IsRegValid:=FALSE;

// Температуры
// Проверка температур
FOR I:=0 TO NUM_TEMPS-1 DO
	IF (pr^.TEMPS[I] < 0) OR (pr^.TEMPS[I] > T_CRITICALS[I]) THEN
		RETURN;
	END_IF
END_FOR

// Температура чиллера
IF (pr^.T_CHIL < 0) OR (pr^.T_CHIL > T_CHIL_CRITICAL) THEN
	RETURN;
END_IF

// Смещение 1-го полупериода
IF pr^.Period.Offsets[0] = pr^.Period.Offsets[1] THEN
	RETURN;
END_IF

// Смещение 2-го полупериода
IF ABS (pr^.Period.Offsets[0] - pr^.Period.Offsets[1]) > WORK_SIZE THEN
	RETURN;
END_IF

// Проценты полупериодов
IF pr^.Period.Per_FirstHP < ASDA_HP_MIN OR pr^.Period.Per_FirstHP > ASDA_HP_MAX THEN
	RETURN;
END_IF

// Проценты импульсов
IF pr^.Period.Per_Pulses[0] < ASDA_PULSE_MIN OR pr^.Period.Per_Pulses[0] > ASDA_PULSE_MAX THEN
	RETURN;
END_IF

IF pr^.Period.Per_Pulses[1] < ASDA_PULSE_MIN OR pr^.Period.Per_Pulses[1] > ASDA_PULSE_MAX THEN
	RETURN;
END_IF

// Проценты уровня
IF pr^.Period.Per_Levels[0] < ASDA_LEVEL_MIN OR pr^.Period.Per_Levels[0] > ASDA_LEVEL_MAX THEN
	RETURN;
END_IF

IF pr^.Period.Per_Levels[1] < ASDA_LEVEL_MIN OR pr^.Period.Per_Levels[1] > ASDA_LEVEL_MAX THEN
	RETURN;
END_IF

// Скорость заготовки
IF pr^.Speed < SPEED_MIN OR pr^.Speed >= SPEED_MAX THEN
	RETURN;
END_IF

// Длина заготовки
IF pr^.Length < LEN_MIN OR pr^.Length > LEN_MAX THEN
	RETURN;
END_IF

// Производительность
IF pr^.Qm < QM_MIN OR pr^.Qm > QM_MAX THEN
	RETURN;
END_IF

IsRegValid:=TRUE;

END_FUNCTION

// Device/Application/SRC/AsdaSetPeriod
PROGRAM AsdaSetPeriod
VAR
	dRep		: DINT;
	wSpeeds		: ARRAY [0..1] OF WORD;			// обороты в мин
	wAccs		: ARRAY [0..3] OF WORD;			// обороты в мин
	wDels		: ARRAY [0..1] OF WORD;			// милисекунды
	dOffsets	: ARRAY [0..1] OF DINT;
	dist		: REAL;
	tPeriod		: REAL;			
	tHalfs		: ARRAY [0..1] OF REAL;
	tPulses		: ARRAY [0..1] OF REAL;
	tLevels		: ARRAY [0..1] OF REAL;
	tAccs		: ARRAY [0..1] OF REAL;
	midSpeeds	: ARRAY [0..1] OF REAL;
	vSpeeds		: ARRAY [0..1] OF REAL;
END_VAR


CASE Asda.SelButton OF

sbPeriod:	// УСТАНОВКА ПАРАМЕТРОВ ПЕРИОДА

	// 1. Сначала записать положение реперной точки P6-01, адрес 16х0602
	dRep:=REAL_TO_DINT (REP_MM * PUU_PER_MM);
	QueuePushReg (ADR (COM1_PRG.WR_REGS), ADR_ASDA, 16#0602, ADR (dRep), 2);			// Р6-01 Положение реперной точки

	// 2. Запись перемещения 1-го полупериода, т.к. оно используется при вычислении следующих параметров
	dOffsets[0]:=REAL_TO_DINT (REG_W.Period.Offsets[0] * PUU_PER_MM);
	QueuePushReg (ADR (COM1_PRG.WR_REGS), ADR_ASDA, 16#062A, ADR (dOffsets[0]), 2);	// Р6-21 Смещение 1-го полупериода рабочее
	QueuePushReg (ADR (COM1_PRG.WR_REGS), ADR_ASDA, 16#063A, ADR (dOffsets[0]), 2);	// Р6-29 Смещение 1-го полупериода для ШАГА позиционирования 14 (ручное перемещение)

	// Запись перемещения 2-го полупериода, т.к. оно используется при вычислении следующих параметров
	dOffsets[1]:=REAL_TO_DINT (REG_W.Period.Offsets[1] * PUU_PER_MM);
	QueuePushReg (ADR (COM1_PRG.WR_REGS), ADR_ASDA, 16#062E, ADR (dOffsets[1]), 2);	// Р6-23 Смещение 2-го полупериода
	QueuePushReg (ADR (COM1_PRG.WR_REGS), ADR_ASDA, 16#063E, ADR (dOffsets[1]), 2);	// Р6-31 Смещение 2-го полупериода для шага позиционирования 15 (ручное перемещение)

	// Время периода в секундах
	tPeriod:= 1 / REG_W.Period.Freq;
	
	// Времена полупериодов в секундах
	tHalfs[0]:=tPeriod * REG_W.Period.Per_FirstHP / 100;
	tHalfs[1]:=tPeriod - tHalfs[0];
	
	// Времена импульсов в секундах
	tPulses[0]:=tHalfs[0] * REG_W.Period.Per_Pulses[0] / 100;
	tPulses[1]:=tHalfs[1] * REG_W.Period.Per_Pulses[1] / 100;
	
	// Фронты полупериодов (импульсов) в секундах - Длина импульса минус длина уровня, делённая на 2
	tAccs[0]:=tPulses[0] * (100 - REG_W.Period.Per_Levels[0]) / 200;
	tAccs[1]:=tPulses[1] * (100 - REG_W.Period.Per_Levels[1]) / 200;
	
	// Уровни полупериодов
	tLevels[0]:=tPulses[0] * REG_W.Period.Per_Levels[0] / 100;
	tLevels[1]:=tPulses[1] * REG_W.Period.Per_Levels[1] / 100;
	
	// Пройденный путь в мм
	dist:=ABS (REG_W.Period.Offsets[0] - REG_W.Period.Offsets[1]);
	
	// Средние скорости в мм/сек
	midSpeeds[0]:=dist / tPulses[0];
	midSpeeds[1]:=dist / tPulses[1];
	
	// Расчётные скорости в мм/сек
	vSpeeds[0]:=midSpeeds[0] * (2 * tAccs[0] + tLevels[0]) / (tAccs[0] + tLevels[0]);
	vSpeeds[1]:=midSpeeds[1] * (2 * tAccs[1] + tLevels[1]) / (tAccs[1] + tLevels[1]);
		
	// Пересчёт скорости, данные - l оборот => 5 мм перемещения
	// 5 мм/сек = 1 об/сек =>
	wSpeeds[0]:=REAL_TO_WORD (vSpeeds[0] * 60 * 10 / 5);	// Получили в об/мин (Нужно умножить на 10, т.к. в сервоприводе единица измерения скорости 0.1 об/мин)
	wSpeeds[1]:=REAL_TO_WORD (vSpeeds[1] * 60 * 10 / 5);	// Получили в об/мин

	// Пересчёт фронт и спада относительно скорости wSpeeds[0]
	wAccs[0]:=REAL_TO_WORD (tAccs[0] * 3000 * 1000 / wSpeeds[0]);	
	wAccs[1]:=REAL_TO_WORD (tAccs[0] * 3000 * 1000 / wSpeeds[0]);
	wAccs[2]:=REAL_TO_WORD (tAccs[1] * 3000 * 1000 / wSpeeds[1]);
	wAccs[3]:=REAL_TO_WORD (tAccs[1] * 3000 * 1000 / wSpeeds[1]);
	
	// Задержки в миллисекундах
	wDels[0]:=REAL_TO_WORD ((tHalfs[0] - tPulses[0]) * 1000.0);
	wDels[1]:=REAL_TO_WORD ((tHalfs[1] - tPulses[1]) * 1000.0);

	// Запись	
	QueuePushReg (ADR (COM1_PRG.WR_REGS), ADR_ASDA, 16#0528, ADR (wAccs[0]), 1);		// Р5-20 Фронт 1-го полупериода
	QueuePushReg (ADR (COM1_PRG.WR_REGS), ADR_ASDA, 16#052A, ADR (wAccs[1]), 1);		// Р5-21 Спад 1-го полупериода 
	QueuePushReg (ADR (COM1_PRG.WR_REGS), ADR_ASDA, 16#052C, ADR (wAccs[2]), 1);		// Р5-22 Фронт 2-го полупериода
	QueuePushReg (ADR (COM1_PRG.WR_REGS), ADR_ASDA, 16#052E, ADR (wAccs[3]), 1);		// Р5-23 Спад 2-го полупериода 

	QueuePushReg (ADR (COM1_PRG.WR_REGS), ADR_ASDA, 16#0578, ADR (wSpeeds[0]), 1);		// Р5-60 Скорость 1-го полупериода
	QueuePushReg (ADR (COM1_PRG.WR_REGS), ADR_ASDA, 16#057A, ADR (wSpeeds[1]), 1);		// Р5-61 Скорость 2-го полупериода 

	QueuePushReg (ADR (COM1_PRG.WR_REGS), ADR_ASDA, 16#0550, ADR (wDels[0]), 1);		// Р5-40 Задержка 1-го полупериода
	QueuePushReg (ADR (COM1_PRG.WR_REGS), ADR_ASDA, 16#0552, ADR (wDels[1]), 1);		// Р5-41 Задержка 2-го полупериода

// Команда Homing
sbHoming: AddWriteCmd (wCmd:=wcAsda_Homing);
	
// Движение вперёд
sbForward: AddWriteCmd (wCmd:=wcAsda_Forward);

// Движение назад
sbBackward: AddWriteCmd (wCmd:=wcAsda_Backward);

// Парковка
sbParking: AddWriteCmd (wCmd:=wcAsda_Parking);

// Работа (пульсирование)
sbWorking: AddWriteCmd (wCmd:=wcAsda_Working);
	
END_CASE

Asda.SelButton:=sbNo;
Asda.bCmd:=FALSE;

END_PROGRAM

// Device/Application/SRC_AUX/SWAP_BYTES
FUNCTION SWAP_BYTES : WORD
VAR_INPUT
	wValue : WORD;
END_VAR
VAR
END_VAR


SWAP_BYTES := SHL (wValue, 8) OR SHR (wValue, 8);

END_FUNCTION

// Device/Application/SRC/SET_FRAME_INDEX_EX
FUNCTION SET_FRAME_INDEX_EX : BYTE
VAR_INPUT
	Index : BYTE;
END_VAR
VAR
END_VAR
VAR // added by the converter: edge detectors and wires of the graphical bodies
    _w1 : ANY;
END_VAR

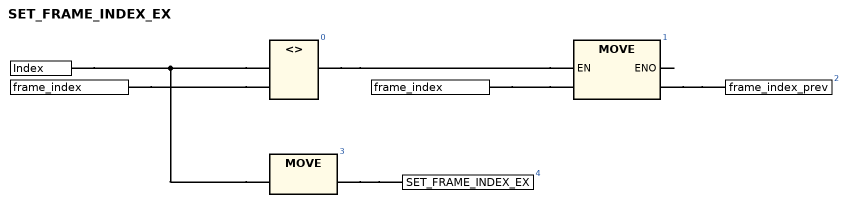
IF Index <> frame_index THEN _w1 := frame_index; END_IF
frame_index_prev := _w1;
SET_FRAME_INDEX_EX := Index;

END_FUNCTION

// Device/Application/SRC_AUX/BYTES_FROM_DINT
FUNCTION BYTES_FROM_DINT : BOOL
VAR_INPUT
	pBytes	: POINTER TO BYTE;
	iDint	: DINT;
END_VAR
VAR
	pB		: POINTER TO BYTE;
END_VAR

BYTES_FROM_DINT:=TRUE;

pB:=ADR(iDint);

pBytes[0]:=pB[1];
pBytes[1]:=pB[0];
pBytes[2]:=pB[3];
pBytes[3]:=pB[2];

END_FUNCTION

// Device/Application/SRC/MERGE_RGB
FUNCTION MERGE_RGB : DWORD
VAR_INPUT
	clR	: BYTE;
	clG	: BYTE;
	clB	: BYTE;
END_VAR
VAR
END_VAR

MERGE_RGB:=BYTE_TO_DWORD(255);
MERGE_RGB:=SHL(MERGE_RGB,8);
MERGE_RGB:=MERGE_RGB OR BYTE_TO_DWORD(clR);
MERGE_RGB:=SHL(MERGE_RGB,8);
MERGE_RGB:=MERGE_RGB OR BYTE_TO_DWORD(clG);
MERGE_RGB:=SHL(MERGE_RGB,8);
MERGE_RGB:=MERGE_RGB OR BYTE_TO_DWORD(clB);

END_FUNCTION

// Device/Application/SRC_FILE/WRITE_OPTIONS
FUNCTION WRITE_OPTIONS : BOOL
VAR_INPUT
	Show	: BOOL;
END_VAR
VAR
	hFile	: SysFile.RTS_IEC_HANDLE;	
	Result	: SysFile.RTS_IEC_RESULT;
	rSize	: __XWORD;
	wrBytes	: __XWORD;
	
END_VAR

WRITE_OPTIONS:=FALSE;
// Создаём новый файл
hFile:=SysFileOpen (OPTIONSFILE,SysFile.AM_WRITE, ADR (Result));
IF Result <> 0 THEN
	RETURN;
END_IF

rSize:=SIZEOF (TSetts);

wrBytes:=SysFileWrite(hFile, ADR (Setts), rSize, ADR (Result));
IF (Result=0) AND (wrBytes=rSize) THEN
	WRITE_OPTIONS:=TRUE;
END_IF

SysFileClose (hFile);

END_FUNCTION

// Device/Application/SRC_AUX/HiWord
FUNCTION HiWord : WORD
VAR_INPUT
	dValue	: DINT;
END_VAR	
VAR
	pW		: POINTER TO WORD;
END_VAR

pW:= ADR (dValue);
HiWord:=pW[1];

END_FUNCTION

// Device/Application/SRC_FILE/READ_OPTIONS
FUNCTION READ_OPTIONS : BOOL
VAR
	hFile	: SysFile.RTS_IEC_HANDLE;	
	Result	: SysFile.RTS_IEC_RESULT;
	fSize	: __XWORD;
	rSize	: __XWORD;
	rdBytes	: __XWORD;
	rdSetts	: TSetts;
	
END_VAR

READ_OPTIONS:=FALSE;

rSize:=SIZEOF(TSetts);

hFile:=SysFileOpen (OPTIONSFILE, SysFile.AM_READ, ADR (Result));
IF Result <> 0 THEN
	RETURN;
END_IF

//  Файл существует, проверяем размер файла
fSize:=SysFileGetSizeByHandle (hFile, ADR (Result));
IF Result <> 0 OR fSize <> rSize THEN
	SysFileClose(hFile);
	RETURN;	
END_IF

rdBytes:=SysFileRead(hFile, ADR (rdSetts), rSize, ADR (Result));	
IF Result = 0 AND rdBytes = rSize THEN
	Setts:=rdSetts;
	READ_OPTIONS:=TRUE;
END_IF

SysFileClose(hFile);

END_FUNCTION

// Device/Application/SRC_AUX/LoWord
FUNCTION LoWord : WORD
VAR_INPUT
	dValue	: DINT;
END_VAR
VAR
	pW		: POINTER TO WORD;
END_VAR

pW:= ADR (dValue);
LoWord:=pW[0];

END_FUNCTION

// Device/Application/SRC_AUX/LoByte
FUNCTION LoByte : BYTE
VAR_INPUT
	W	: WORD;
END_VAR
VAR
END_VAR

LoByte:=WORD_TO_BYTE (W AND 16#FF);

END_FUNCTION

// Device/Application/SRC_AUX/HiByte
FUNCTION HiByte : BYTE
VAR_INPUT
	W : WORD;
END_VAR
VAR
END_VAR

HiByte:= WORD_TO_BYTE (SHR (W, 8) AND 16#FF);

END_FUNCTION

// Device/Application/SRC_AUX/IsRegTempersValid
FUNCTION IsRegTempersValid : BOOL
VAR_INPUT
	pr : POINTER TO TReg;
	
END_VAR
VAR
	I: INT;
END_VAR

IsRegTempersValid:=FALSE;

// Температуры
// Проверка температур уставок (без TEMPS[7])	
FOR I:=0 TO NUM_TEMPS-2 DO
	
	// Если задана температура ниже температуры запуска приводов или выше критической 
	IF (pr^.TEMPS[I] < Setts.T_ZAP[I]) OR (pr^.TEMPS[I] > T_CRITICALS[I]) THEN
		RETURN;
	END_IF
	
END_FOR

IsRegTempersValid:=TRUE;

END_FUNCTION

// Device/Application/SRC_AUX/BYTES_FROM_INT
FUNCTION BYTES_FROM_INT : BOOL
VAR_INPUT
	pBytes	: POINTER TO BYTE;
	vInt	: INT;
END_VAR
VAR
	pB		: POINTER TO BYTE;
END_VAR

BYTES_FROM_INT:=TRUE;

pB:=ADR(vInt);
pBytes[0]:=pB[1];
pBytes[1]:=pB[0];

END_FUNCTION

// Device/Application/Visu/VIS_AUX
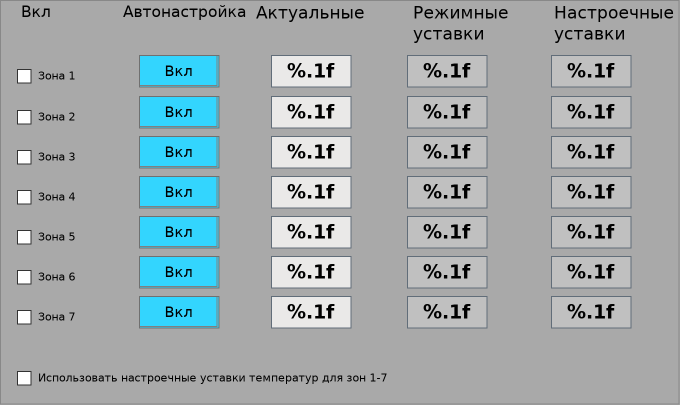
VISUALIZATION VIS_AUX  // 680x405
    Checkbox (15,55 120x42), "Зона 1", variable: Dvp.T_Enables.0
    Checkbox (15,96 120x42), "Зона 2", variable: Dvp.T_Enables.1
    Checkbox (15,136 120x42), "Зона 3", variable: Dvp.T_Enables.2
    Checkbox (15,176 120x42), "Зона 4", variable: Dvp.T_Enables.3
    Checkbox (15,216 120x42), "Зона 5", variable: Dvp.T_Enables.4
    Checkbox (15,256 120x42), "Зона 6", variable: Dvp.T_Enables.5
    Checkbox (15,296 120x42), "Зона 7", variable: Dvp.T_Enables.6
    Label (18,1 63x24), "Вкл"
    Label (120,1 129x28), "Автонастройка"
    Button (139,55 80x32), "Вкл", colour toggle: Dvp.Auto_IN.0
        OnMouseClick: execute { Dvp.Auto_OUT.0:=TRUE; }
    Button (139,96 80x32), "Вкл", colour toggle: Dvp.Auto_IN.1
        OnMouseClick: execute { Dvp.Auto_OUT.1:=TRUE; }
    Button (139,136 80x32), "Вкл", colour toggle: Dvp.Auto_IN.2
        OnMouseClick: execute { Dvp.Auto_OUT.2:=TRUE; }
    Button (139,176 80x32), "Вкл", colour toggle: Dvp.Auto_IN.3
        OnMouseClick: execute { Dvp.Auto_OUT.3:=TRUE; }
    Button (139,216 80x32), "Вкл", colour toggle: Dvp.Auto_IN.4
        OnMouseClick: execute { Dvp.Auto_OUT.4:=TRUE; }
    Button (139,256 80x32), "Вкл", colour toggle: Dvp.Auto_IN.5
        OnMouseClick: execute { Dvp.Auto_OUT.5:=TRUE; }
    Button (139,296 80x32), "Вкл", colour toggle: Dvp.Auto_IN.6
        OnMouseClick: execute { Dvp.Auto_OUT.6:=TRUE; }
    Checkbox (15,357 589x42), "Использовать настроечные уставки температур для зон 1-7", variable: zd_selector
    RoundedRectangle (407,55 80x32), "%.1f", text variable: REG_W.TEMPS[0], colour toggle: NOT zd_selector
    RoundedRectangle (407,96 80x32), "%.1f", text variable: REG_W.TEMPS[1], colour toggle: NOT zd_selector
    RoundedRectangle (407,136 80x32), "%.1f", text variable: REG_W.TEMPS[2], colour toggle: NOT zd_selector
    RoundedRectangle (407,176 80x32), "%.1f", text variable: REG_W.TEMPS[3], colour toggle: NOT zd_selector
    RoundedRectangle (407,216 80x32), "%.1f", text variable: REG_W.TEMPS[4], colour toggle: NOT zd_selector
    RoundedRectangle (407,256 80x32), "%.1f", text variable: REG_W.TEMPS[5], colour toggle: NOT zd_selector
    RoundedRectangle (407,296 80x32), "%.1f", text variable: REG_W.TEMPS[6], colour toggle: NOT zd_selector
    Label (410,1 107x49), "Режимные уставки"
    RoundedRectangle (551,55 80x32), "%.1f", text variable: zd_temps[0], colour toggle: zd_selector
        OnMouseClick: write the text variable via VisuDialogs.Numpad, min T_MINS_ZAD[6], max T_MAXS_ZAD[6], title "ТЕМПЕРАТУРА 7 ЗОНЫ"
    RoundedRectangle (551,96 80x32), "%.1f", text variable: zd_temps[1], colour toggle: zd_selector
        OnMouseClick: write the text variable via VisuDialogs.Numpad, min T_MINS_ZAD[0], max T_MAXS_ZAD[0]
    RoundedRectangle (551,136 80x32), "%.1f", text variable: zd_temps[2], colour toggle: zd_selector
        OnMouseClick: write the text variable via VisuDialogs.Numpad, min T_MINS_ZAD[0], max T_MAXS_ZAD[0]
    RoundedRectangle (551,176 80x32), "%.1f", text variable: zd_temps[3], colour toggle: zd_selector
        OnMouseClick: write the text variable via VisuDialogs.Numpad, min T_MINS_ZAD[0], max T_MAXS_ZAD[0]
    RoundedRectangle (551,216 80x32), "%.1f", text variable: zd_temps[4], colour toggle: zd_selector
        OnMouseClick: write the text variable via VisuDialogs.Numpad, min T_MINS_ZAD[0], max T_MAXS_ZAD[0]
    RoundedRectangle (551,256 80x32), "%.1f", text variable: zd_temps[5], colour toggle: zd_selector
        OnMouseClick: write the text variable via VisuDialogs.Numpad, min T_MINS_ZAD[0], max T_MAXS_ZAD[0]
    RoundedRectangle (551,296 80x32), "%.1f", text variable: zd_temps[6], colour toggle: zd_selector
        OnMouseClick: write the text variable via VisuDialogs.Numpad, min T_MINS_ZAD[0], max T_MAXS_ZAD[0]
    Label (551,1 127x47), "Настроечные уставки"
    RoundedRectangle (271,55 80x32), "%.1f", text variable: Dvp.T_Actuals[0], colour variable: Dvp.FillColors[0]
        p3450524324: Dvp.FrameColors[0]
    RoundedRectangle (271,96 80x32), "%.1f", text variable: Dvp.T_Actuals[1], colour variable: Dvp.FillColors[1]
        p3450524324: Dvp.FrameColors[1]
    RoundedRectangle (271,136 80x32), "%.1f", text variable: Dvp.T_Actuals[2], colour variable: Dvp.FillColors[2]
        p3450524324: Dvp.FrameColors[2]
    RoundedRectangle (271,176 80x32), "%.1f", text variable: Dvp.T_Actuals[3], colour variable: Dvp.FillColors[3]
        p3450524324: Dvp.FrameColors[3]
    RoundedRectangle (271,216 80x32), "%.1f", text variable: Dvp.T_Actuals[4], colour variable: Dvp.FillColors[4]
        p3450524324: Dvp.FrameColors[4]
    RoundedRectangle (271,256 80x32), "%.1f", text variable: Dvp.T_Actuals[5], colour variable: Dvp.FillColors[5]
        p3450524324: Dvp.FrameColors[5]
    RoundedRectangle (271,296 80x32), "%.1f", text variable: Dvp.T_Actuals[6], colour variable: Dvp.FillColors[6]
        p3450524324: Dvp.FrameColors[6]
    Label (249,1 123x32), "Актуальные"
END_VISUALIZATION

// Device/Application/Visu/Main_Panel
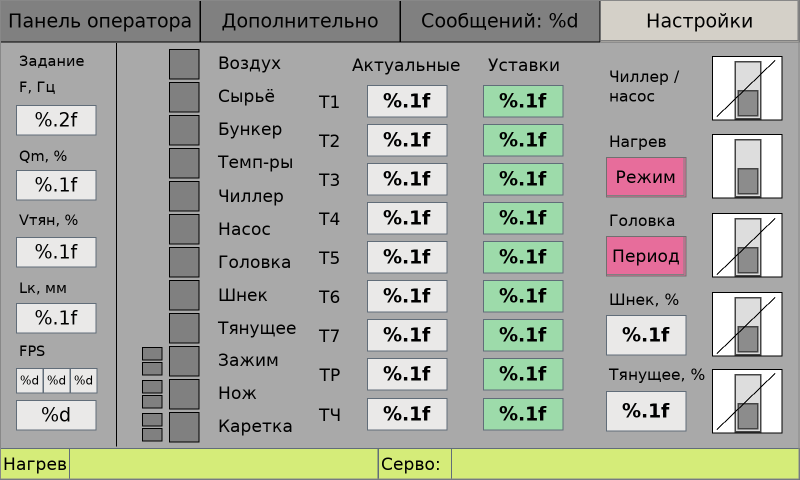
VISUALIZATION Main_Panel  // 800x480
    Rectangle (0,448 80x32), "Нагрев:"
    Frame (118,43 692x442), frame switch variable: frame_index
        shows VIS_OPERATOR()
        shows VIS_AUX()
        shows VIS_MSGS()
        shows VIS_PERIOD()
        shows VIS_REG()
    Label (16,77 48x25), "F, Гц"
    RoundedRectangle (16,170 80x30), "%.1f", text variable: Shnek.Qm
    Label (16,146 77x27), "Qm, %"
    Label (16,210 92x26), "Vтян, %"
    RoundedRectangle (16,237 80x30), "%.1f", text variable: Pulling.Speed
    Label (16,278 59x25), "Lк, мм"
    RoundedRectangle (16,303 80x30), "%.1f", text variable: REG_W.Length
    RoundedRectangle (16,105 80x30), "%.2f", text variable: REG_W.Period.Freq
    Label (16,51 79x20), "Задание"
    Line (116,43) (116,446)
    Rectangle (0,0 200x42), "Панель оператора", colour toggle: frame_index=0
        OnMouseClick: execute { SET_FRAME_INDEX (0); }
    Rectangle (200,0 200x42), "Дополнительно", colour toggle: frame_index=1
        OnMouseClick: execute { SET_FRAME_INDEX (1); }
    Rectangle (400,0 200x42), "Сообщений: %d", text variable: alarm_count, colour toggle: frame_index=2
        OnMouseClick: execute { SET_FRAME_INDEX (2); }
    Button (600,0 200x42), "Настройки"
        OnMouseClick:  Assign=Setts_Panel, Type=Assignment
    Rectangle (69,448 309x32), text list: 'DvpTextList', text index: Dvp.text_id
    Rectangle (378,448 80x32), "Серво:"
    Rectangle (451,448 349x32), text list: 'AsdaTextList', text index: Asda.text_id
    RoundedRectangle (16,400 80x30), "%d", text variable: FPS_FULL
    Label (16,341 59x25), "FPS"
    RoundedRectangle (16,368 27x25), "%d", text variable: COM1_PRG.FPS
    RoundedRectangle (43,368 27x25), "%d", text variable: COM2_PRG.FPS
    RoundedRectangle (70,368 27x25), "%d", text variable: COM3_PRG.FPS
END_VISUALIZATION

// Device/Application/Visu/DlgConfirm
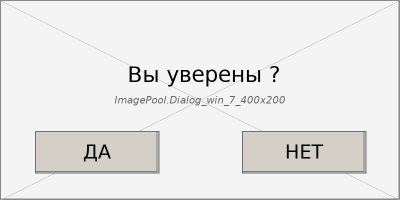
VISUALIZATION DlgConfirm  // 400x200
VAR_IN_OUT
	bDialogVar	: BOOL;
END_VAR
    Image (0,0 400x200), image: ImagePool.Dialog_win_7_400x200
    Button (35,131 124x42), "ДА"
        OnMouseClick:  Dialog=DlgConfirm, Result=OK, NumpadKeypadSet=True
        OnMouseClick: execute { bDialogVar:=TRUE; }
    Button (242,131 124x42), "НЕТ"
        OnMouseClick:  Dialog=DlgConfirm, Result=Cancel, NumpadKeypadSet=True
    Label (80,55 248x39), "Вы уверены ?"
END_VISUALIZATION

// Device/Application/Visu/Panel_Reg
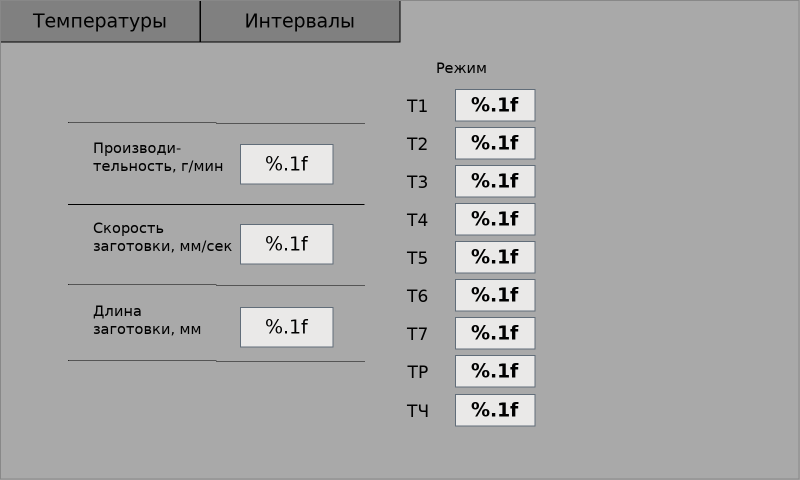
VISUALIZATION Panel_Reg  // 800x480
    Frame (6,47 734x398), frame switch variable: frame_index_reg
        shows VIS_REG()
        shows VIS_PERIOD()
    Rectangle (0,0 200x42), "Температуры", colour toggle: frame_index_reg=0
        OnMouseClick: execute { frame_index_reg:=0; }
    Rectangle (200,0 200x42), "Интервалы", colour toggle: frame_index_reg=1
        OnMouseClick: execute { frame_index_reg:=1; }
END_VISUALIZATION

// Device/Application/Visu/VIS_MSGS
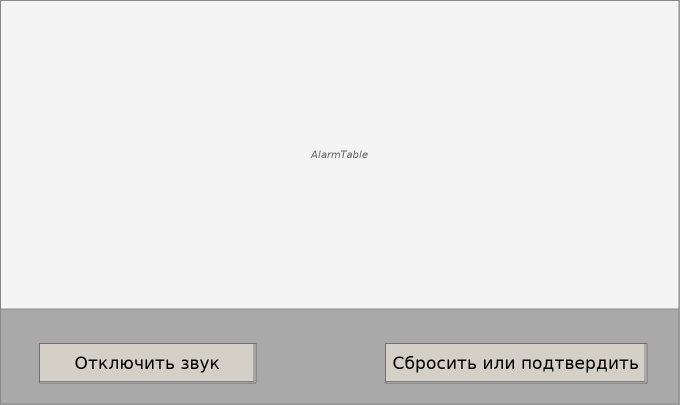
VISUALIZATION VIS_MSGS  // 680x405
    AlarmTable (0,0 679x309)
        Column[0]: ColumnTitle=Сигнал
        Column[1]: ColumnTitle=Сообщение
        p1521930926: __All
        p1663851261: __All
        p1347137028: alarm_count
    Button (385,343 262x40), "Сбросить или подтвердить"
        OnMouseClick: execute { ALARM_RESET:=TRUE; }
    Button (39,343 217x40), "Отключить звук", colour toggle: Dvp.ALARM_ZVUK AND NOT Setts.otkl_alarm_zvuk
        OnMouseClick: execute { Dvp.ALARM_ZVUK:=FALSE; }
END_VISUALIZATION

// Device/Application/Visu/Setts_Panel
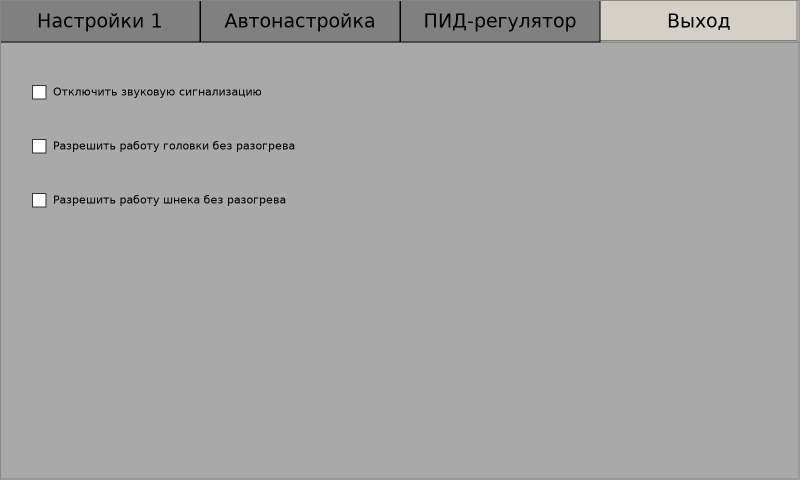
VISUALIZATION Setts_Panel  // 800x480
    Button (599,0 200x42), "Выход"
        OnMouseClick:  Assign=Main_Panel, Type=Assignment
    Rectangle (0,0 200x42), "Настройки 1", colour toggle: frame_index_setts=0
        OnMouseClick: execute { frame_index_setts:=0; }
    Rectangle (200,0 200x42), "Автонастройка", colour toggle: frame_index_setts=1
        OnMouseClick: execute { frame_index_setts:=1; }
    Rectangle (400,0 200x42), "ПИД-регулятор", colour toggle: frame_index_setts=2
        OnMouseClick: execute { frame_index_setts:=2; }
    Frame (0,43 793x430)
        shows VIS_SETTS_1()
        shows VIS_SETTS_2()
        shows VIS_SETTS_3()
END_VISUALIZATION

// Device/Application/Visu/VIS_REG
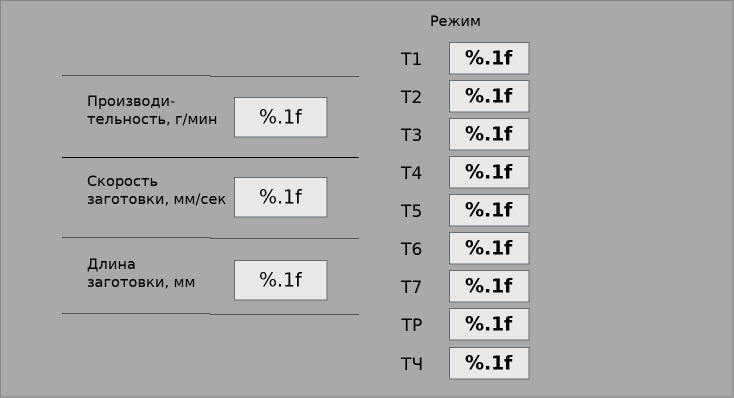
VISUALIZATION VIS_REG  // 734x398
    Line (62,313) (358,314)
    Line (62,237) (358,238)
    Line (62,157) (358,157)
    Line (62,75) (358,76)
    Label (84,91 162x53), "Производи- тельность, г/мин"
    Label (84,171 167x50), "Скорость заготовки, мм/сек"
    RoundedRectangle (234,177 93x40), "%.1f", text variable: REG_W.Speed
        OnMouseClick: write the text variable via VisuDialogs.Numpad, min SPEED_MIN, max SPEED_MAX, title "Скорость заготовки, мм/сек"
    Label (84,254 126x53), "Длина заготовки, мм"
    RoundedRectangle (234,260 93x40), "%.1f", text variable: REG_W.Length
        OnMouseClick: write the text variable via VisuDialogs.Numpad, min LEN_MIN, max LEN_MAX, title "Длина заготовки, мм"
    RoundedRectangle (449,42 80x32), "%.1f", text variable: REG_W.TEMPS[0]
        OnMouseClick: write the text variable via VisuDialogs.Numpad, min T_MINS_ZAD[0], max T_MAXS_ZAD[0], title "ТЕМПЕРАТУРА 1 ЗОНЫ"
    Label (392,43 40x32), "T1"
    RoundedRectangle (449,80 80x32), "%.1f", text variable: REG_W.TEMPS[1]
        OnMouseClick: write the text variable via VisuDialogs.Numpad, min T_MINS_ZAD[1], max T_MAXS_ZAD[1], title "ТЕМПЕРАТУРА 2 ЗОНЫ"
    Label (392,81 40x32), "T2"
    RoundedRectangle (449,118 80x32), "%.1f", text variable: REG_W.TEMPS[2]
        OnMouseClick: write the text variable via VisuDialogs.Numpad, min T_MINS_ZAD[2], max T_MAXS_ZAD[2], title "ТЕМПЕРАТУРА3 ЗОНЫ"
    Label (392,119 40x32), "T3"
    RoundedRectangle (449,156 80x32), "%.1f", text variable: REG_W.TEMPS[3]
        OnMouseClick: write the text variable via VisuDialogs.Numpad, min T_MINS_ZAD[3], max T_MAXS_ZAD[3], title "ТЕМПЕРАТУРА 4 ЗОНЫ"
    Label (392,157 40x32), "T4"
    RoundedRectangle (449,194 80x32), "%.1f", text variable: REG_W.TEMPS[4]
        OnMouseClick: write the text variable via VisuDialogs.Numpad, min T_MINS_ZAD[4], max T_MAXS_ZAD[4], title "ТЕМПЕРАТУРА 5 ЗОНЫ"
    Label (392,195 40x32), "T5"
    RoundedRectangle (449,232 80x32), "%.1f", text variable: REG_W.TEMPS[5]
        OnMouseClick: write the text variable via VisuDialogs.Numpad, min T_MINS_ZAD[5], max T_MAXS_ZAD[5], title "ТЕМПЕРАТУРА 6 ЗОНЫ"
    Label (392,233 40x32), "T6"
    RoundedRectangle (449,270 80x32), "%.1f", text variable: REG_W.TEMPS[6]
        OnMouseClick: write the text variable via VisuDialogs.Numpad, min T_MINS_ZAD[6], max T_MAXS_ZAD[6], title "ТЕМПЕРАТУРА 7 ЗОНЫ"
    Label (392,271 40x32), "T7"
    RoundedRectangle (449,308 80x32), "%.1f", text variable: REG_W.TEMPS[7]
        OnMouseClick: write the text variable via VisuDialogs.Numpad, min T_MINS_ZAD[7], max T_MAXS_ZAD[7], title "ТЕМПЕРАТУРА РАСПЛАВА"
    Label (392,309 40x32), "TР"
    RoundedRectangle (449,347 80x32), "%.1f", text variable: REG_W.T_CHIL
        OnMouseClick: write the text variable via VisuDialogs.Numpad, min T_MIN_CHIL_ZAD, max T_MAX_CHIL_ZAD, title "ТЕМПЕРАТУРА ЧИЛЛЕРА"
    Label (392,348 40x32), "TЧ"
    Label (427,6 76x30), "Режим"
    RoundedRectangle (234,97 93x40), "%.1f", text variable: REG_W.Qm
        OnMouseClick: write the text variable via VisuDialogs.Numpad, min QM_MIN, max QM_MAX, title "Производительность, %"
END_VISUALIZATION

// Device/Application/Visu/VIS_PERIOD
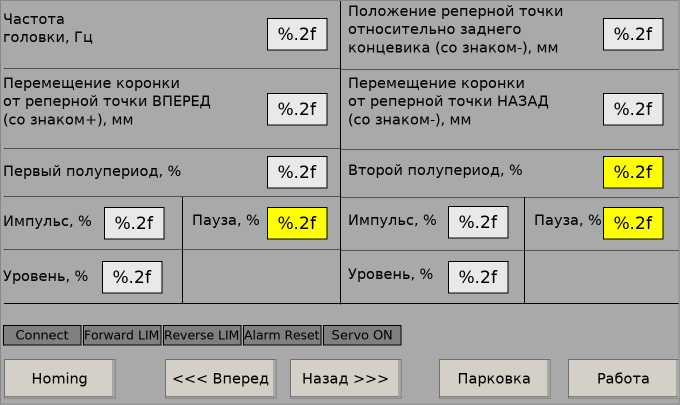
VISUALIZATION VIS_PERIOD  // 680x405
    RoundedRectangle (603,18 60x32), "%.2f", text variable: REP_MM
        OnMouseClick: write the text variable via VisuDialogs.Numpad, min REP_MIN, max REP_MAX, title "ЗАДАТЬ РЕПЕРНУЮ ТОЧКУ"
        OnDialogClosed: execute { Asda.SelButton:=sbPeriod; AsdaSetPeriod (); }
    Button (439,359 111x39), "Парковка", input disabled if: NOT Asda.WAIT
        OnMouseClick:  Dialog=DlgConfirm, Parameters={bDialogVar: Asda.bCmd}, Selected={1: }, OpenModal=True, OpenCentered=True
        OnDialogClosed: execute {
            IF Asda.bCmd THEN
            	Asda.SelButton:=sbParking;
            	AsdaSetPeriod ();
            END_IF
        }
    Label (345,1 220x69), "Положение реперной точки относительно заднего концевика (со знаком-), мм"
    Label (0,266 102x25), "Уровень, %"
    RoundedRectangle (102,261 60x32), "%.2f", text variable: REG_W.Period.Per_Levels[0]
        OnMouseClick: write the text variable via VisuDialogs.Numpad, min ASDA_LEVEL_MIN, max ASDA_LEVEL_MAX, title "УРОВЕНЬ ПЕРВОГО П/П"
        OnDialogClosed: execute { Asda.SelButton:=sbPeriod; AsdaSetPeriod (); }
    RoundedRectangle (448,261 60x32), "%.2f", text variable: REG_W.Period.Per_Levels[1]
        OnMouseClick: write the text variable via VisuDialogs.Numpad, min ASDA_LEVEL_MIN, max ASDA_LEVEL_MAX, title "УРОВЕНЬ ВТОРОГО П/П"
        OnDialogClosed: execute { Asda.SelButton:=sbPeriod; AsdaSetPeriod (); }
    Label (0,73 251x72), "Перемещение коронки от реперной точки ВПЕРЕД (со знаком+), мм"
    RoundedRectangle (267,93 60x32), "%.2f", text variable: REG_W.Period.Offsets[0]
        OnMouseClick: write the text variable via VisuDialogs.Numpad, min REP_MM + 0.3, max WORK_SIZE + REP_MM - 0.3, title "ПЕРЕМЕЩЕНИЕ 1-ГО П/П"
        OnDialogClosed: execute { Asda.SelButton:=sbPeriod; AsdaSetPeriod (); }
    Label (345,73 233x71), "Перемещение коронки от реперной точки НАЗАД (со знаком-), мм"
    RoundedRectangle (603,93 60x32), "%.2f", text variable: REG_W.Period.Offsets[1]
        OnMouseClick: write the text variable via VisuDialogs.Numpad, min REP_MM + 0.3, max WORK_SIZE + REP_MM - 0.3, title "ПЕРЕМЕЩЕНИЕ 2-ГО П/П"
        OnDialogClosed: execute { Asda.SelButton:=sbPeriod; AsdaSetPeriod (); }
    Button (568,359 111x39), "Работа", input disabled if: NOT Asda.WAIT
        OnMouseClick:  Dialog=DlgConfirm, Parameters={bDialogVar: Asda.bCmd}, Selected={1: }, OpenModal=True, OpenCentered=True
        OnDialogClosed: execute {
            IF Asda.bCmd THEN
            	Asda.SelButton:=sbWorking;
            	AsdaSetPeriod ();
            END_IF
        }
    Button (4,359 111x39), "Homing", input disabled if: NOT Asda.WAIT
        OnMouseClick:  Dialog=DlgConfirm, Parameters={bDialogVar: Asda.bCmd}, Selected={1: }, OpenModal=True, OpenCentered=True
        OnDialogClosed: execute {
            IF Asda.bCmd THEN
            	Asda.SelButton:=sbHoming;
            	AsdaSetPeriod ();
            END_IF
        }
    Button (165,359 111x39), "<<< Вперед", input disabled if: NOT Asda.WAIT
        OnMouseClick:  Dialog=DlgConfirm, Parameters={bDialogVar: Asda.bCmd}, Selected={1: }, OpenModal=True, OpenCentered=True
        OnDialogClosed: execute {
            IF Asda.bCmd THEN
            	Asda.SelButton:=sbForward;
            	AsdaSetPeriod ();
            END_IF
        }
    Button (290,359 111x39), "Назад >>>", input disabled if: NOT Asda.WAIT
        OnMouseClick:  Dialog=DlgConfirm, Parameters={bDialogVar: Asda.bCmd}, Selected={1: }, OpenModal=True, OpenCentered=True
        OnDialogClosed: execute {
            IF Asda.bCmd THEN
            	Asda.SelButton:=sbBackward;
            	AsdaSetPeriod ();
            END_IF
        }
    Line (4,68) (678,69)
    Line (4,303) (678,303)
    Line (4,196) (678,197)
    Label (0,161 214x23), "Первый полупериод, %"
    Label (345,160 216x23), "Второй полупериод, %"
    Label (345,264 97x25), "Уровень, %"
    Line (340,0) (340,304)
    RoundedRectangle (267,156 60x32), "%.2f", text variable: REG_W.Period.Per_FirstHP
        OnMouseClick: write the text variable via VisuDialogs.Numpad, min ASDA_HP_MIN, max ASDA_HP_MAX, title "ПЕРВЫЙ ПОЛУПЕРИОД"
        OnDialogClosed: execute { Asda.SelButton:=sbPeriod; AsdaSetPeriod (); }
    RoundedRectangle (603,156 60x32), "%.2f", text variable: 100 - REG_W.Period.Per_FirstHP
    Line (4,249) (678,250)
    Line (182,197) (182,303)
    RoundedRectangle (104,207 60x32), "%.2f", text variable: REG_W.Period.Per_Pulses[0]
        OnMouseClick: write the text variable via VisuDialogs.Numpad, min ASDA_PULSE_MIN, max ASDA_PULSE_MAX, title "ПЕРВЫЙ ПОЛУПЕРИОД"
        OnDialogClosed: execute { Asda.SelButton:=sbPeriod; AsdaSetPeriod (); }
    Label (0,211 94x23), "Импульс, %"
    Label (189,210 94x23), "Пауза, %"
    RoundedRectangle (267,207 60x32), "%.2f", text variable: 100-REG_W.Period.Per_Pulses[0]
    Label (345,210 94x23), "Импульс, %"
    RoundedRectangle (448,206 60x32), "%.2f", text variable: REG_W.Period.Per_Pulses[1]
        OnMouseClick: write the text variable via VisuDialogs.Numpad, min ASDA_PULSE_MIN, max ASDA_PULSE_MAX, title "ПЕРВЫЙ ПОЛУПЕРИОД"
        OnDialogClosed: execute { Asda.SelButton:=sbPeriod; AsdaSetPeriod (); }
    Label (531,210 94x23), "Пауза, %"
    RoundedRectangle (603,207 60x32), "%.2f", text variable: 100-REG_W.Period.Per_Pulses[1]
    Line (524,197) (524,303)
    Line (4,148) (678,149)
    RoundedRectangle (3,325 78x20), "Connect", colour toggle: Asda.Connect
    RoundedRectangle (243,325 78x20), "Alarm Reset", colour toggle: Asda.P4_07.1
    RoundedRectangle (323,325 78x20), "Servo ON", colour toggle: Asda.P4_07.0
    RoundedRectangle (163,325 78x20), "Reverse LIM", colour toggle: Asda.P4_07.2
    RoundedRectangle (83,325 78x20), "Forward LIM", colour toggle: Asda.P4_07.3
    Label (0,9 144x54), "Частота головки, Гц"
    RoundedRectangle (267,18 60x32), "%.2f", text variable: REG_W.Period.Freq
        OnMouseClick: write the text variable via VisuDialogs.Numpad, min FREQ_MIN, max FREQ_MAX, title "ЧАСТОТА ГОЛОВКИ, Гц"
        OnDialogClosed: execute {
            //VisuDialogs.Numpad_VISU_STRUCT.bInit
            Asda.SelButton:=sbPeriod;
            AsdaSetPeriod ();
        }
END_VISUALIZATION

// Device/Application/Visu/VIS_OPERATOR
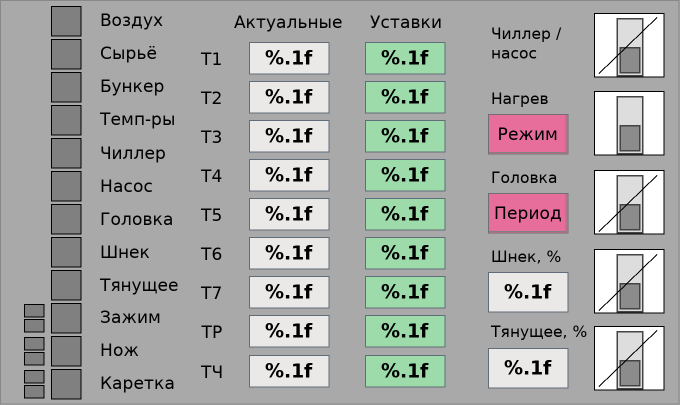
VISUALIZATION VIS_OPERATOR  // 680x405
    RoundedRectangle (594,91 70x64), colour variable: Dvp.NagrevFillColor
        p3450524324: Dvp.NagrevFrameColor
    DipSwitch (601,96 58x58), variable: Dvp.Nagrev_on, behaviour: TOGGLE, style: Switch-DipSwitch-Gray
    RoundedRectangle (594,326 70x64), colour variable: Pulling.BtnFillColor
        p3450524324: Pulling.BtnFrameColor
    DipSwitch (601,331 58x58), variable: Pulling.Pusk, input disabled if: Pulling.Block, behaviour: TOGGLE, style: Switch-DipSwitch-Gray
    RoundedRectangle (594,249 70x64), colour variable: Shnek.FillColor
        p3450524324: Shnek.FrameColor
    DipSwitch (601,254 58x58), variable: Shnek.Pusk, input disabled if: Shnek.Block, behaviour: TOGGLE, style: Switch-DipSwitch-Gray
    RoundedRectangle (594,170 70x64), colour variable: Asda.BtnFillColor
        p3450524324: Asda.BtnFrameColor
    DipSwitch (601,175 58x58), variable: Asda.Pusk, input disabled if: Asda.Block, behaviour: TOGGLE, style: Switch-DipSwitch-Gray
    RoundedRectangle (249,42 80x32), "%.1f", text variable: Dvp.T_Actuals[0], colour variable: Dvp.FillColors[0]
        p3450524324: Dvp.FrameColors[0]
    Label (192,43 40x32), "T1"
    RoundedRectangle (365,42 80x32), "%.1f", text variable: REG_W.TEMPS[0], colour toggle: Dvp.Auto_IN.0
    RoundedRectangle (365,81 80x32), "%.1f", text variable: REG_W.TEMPS[1], colour toggle: Dvp.Auto_IN.1
    RoundedRectangle (249,81 80x32), "%.1f", text variable: Dvp.T_Actuals[1], colour variable: Dvp.FillColors[1]
        p3450524324: Dvp.FrameColors[1]
    Label (192,82 40x32), "T2"
    RoundedRectangle (365,120 80x32), "%.1f", text variable: REG_W.TEMPS[2], colour toggle: Dvp.Auto_IN.2
    RoundedRectangle (249,120 80x32), "%.1f", text variable: Dvp.T_Actuals[2], colour variable: Dvp.FillColors[2]
        p3450524324: Dvp.FrameColors[2]
    Label (192,121 40x32), "T3"
    RoundedRectangle (365,159 80x32), "%.1f", text variable: REG_W.TEMPS[3], colour toggle: Dvp.Auto_IN.3
    RoundedRectangle (249,159 80x32), "%.1f", text variable: Dvp.T_Actuals[3], colour variable: Dvp.FillColors[3]
        p3450524324: Dvp.FrameColors[3]
    Label (192,160 40x32), "T4"
    RoundedRectangle (365,198 80x32), "%.1f", text variable: REG_W.TEMPS[4], colour toggle: Dvp.Auto_IN.4
    RoundedRectangle (249,198 80x32), "%.1f", text variable: Dvp.T_Actuals[4], colour variable: Dvp.FillColors[4]
        p3450524324: Dvp.FrameColors[4]
    Label (192,199 40x32), "T5"
    RoundedRectangle (365,237 80x32), "%.1f", text variable: REG_W.TEMPS[5], colour toggle: Dvp.Auto_IN.5
    RoundedRectangle (249,237 80x32), "%.1f", text variable: Dvp.T_Actuals[5], colour variable: Dvp.FillColors[5]
        p3450524324: Dvp.FrameColors[5]
    Label (192,238 40x32), "T6"
    RoundedRectangle (365,276 80x32), "%.1f", text variable: REG_W.TEMPS[6], colour toggle: Dvp.Auto_IN.6
    RoundedRectangle (249,276 80x32), "%.1f", text variable: Dvp.T_Actuals[6], colour variable: Dvp.FillColors[6]
        p3450524324: Dvp.FrameColors[6]
    Label (192,277 40x32), "T7"
    RoundedRectangle (365,315 80x32), "%.1f", text variable: REG_W.TEMPS[7]
    RoundedRectangle (249,315 80x32), "%.1f", text variable: Dvp.T_Actuals[7], colour variable: Dvp.FillColors[7]
        p3450524324: Dvp.FrameColors[7]
    Label (192,316 40x32), "TР"
    RoundedRectangle (365,355 80x32), "%.1f", text variable: REG_W.T_CHIL
    RoundedRectangle (249,355 80x32), "%.1f", text variable: Chiller.T_ACTUAL, colour variable: Chiller.FillColor
        p3450524324: Chiller.FrameColor
    Label (192,356 40x32), "TЧ"
    RoundedRectangle (51,105 30x30), colour toggle: Dvp.temper_reached
    Label (97,103 89x32), "Tемп-ры"
    RoundedRectangle (51,204 30x30), colour toggle: Asda.Pusk
    Label (97,203 89x32), "Головка"
    RoundedRectangle (51,237 30x30), colour toggle: Shnek.Pusk
    Label (97,236 89x32), "Шнек"
    RoundedRectangle (51,270 30x30), colour toggle: Pulling.Pusk
    Label (97,269 89x32), "Тянущее"
    RoundedRectangle (51,6 30x30), colour toggle: Dvp.PVozd_si
    Label (97,4 89x32), "Воздух"
    RoundedRectangle (51,171 30x30), colour toggle: Dvp.Nasos_si
    Label (97,170 89x32), "Насос"
    RoundedRectangle (51,39 30x30), colour toggle: Dvp.Uroven_si
    Label (97,37 89x32), "Сырьё"
    RoundedRectangle (51,72 30x30), colour toggle: Dvp.Bunker_si
    Label (97,70 89x32), "Бункер"
    RoundedRectangle (594,13 70x64), colour variable: Chiller.BtnFillColor
        p3450524324: Chiller.BtnFrameColor
    DipSwitch (601,18 58x58), variable: Chiller.Pusk, input disabled if: Chiller.Block, behaviour: TOGGLE, style: Switch-DipSwitch-Gray
    Label (488,22 103x43), "Чиллер / насос"
    Line (599,310) (657,254), invisible if: NOT Shnek.Block
    Line (599,386) (657,330), invisible if: NOT Pulling.Block
    Line (599,231) (657,175), invisible if: NOT Asda.Block
    Line (599,73) (657,17), invisible if: NOT Chiller.Block
    RoundedRectangle (51,138 30x30), colour toggle: Chiller.Connect
    Label (97,137 89x32), "Чиллер"
    Button (488,114 80x40), "Режим"
        OnMouseClick: execute { SET_FRAME_INDEX (4); }
    Label (488,88 91x33), "Нагрев"
    Button (488,193 80x40), "Период"
        OnMouseClick: execute { SET_FRAME_INDEX (3); }
    Label (488,167 91x33), "Головка"
    Label (488,246 91x33), "Шнек, %"
    RoundedRectangle (488,348 80x40), "%.1f", text variable: REG_W.Speed
        OnMouseClick: write the text variable via VisuDialogs.Numpad, min SPEED_MIN, max SPEED_MAX, title "Скорость тянущего, %"
    Label (488,321 107x33), "Тянущее, %"
    Label (97,301 89x32), "Зажим"
    RoundedRectangle (51,303 30x30), colour toggle: Dvp.Zazh_si
    Label (97,334 89x32), "Нож"
    RoundedRectangle (51,336 30x30), colour toggle: Dvp.Knife_si
    Label (97,367 89x32), "Каретка"
    RoundedRectangle (51,369 30x30), colour toggle: Dvp.Karet_si
    RoundedRectangle (24,304 20x13), colour toggle: Dvp.ZazhIsx_si
    RoundedRectangle (24,319 20x13), colour toggle: Dvp.ZazhRab_si
    RoundedRectangle (24,337 20x13), colour toggle: Dvp.KnifeIsx_si
    RoundedRectangle (24,352 20x13), colour toggle: Dvp.KnifeRab_si
    RoundedRectangle (24,370 20x13), colour toggle: Dvp.KarIsx_si
    RoundedRectangle (24,385 20x13), colour toggle: Dvp.KarRab_si
    RoundedRectangle (488,272 80x40), "%.1f", text variable: REG_W.Qm
        OnMouseClick: write the text variable via VisuDialogs.Numpad, min QM_MIN, max QM_MAX, title "Производительность, %"
    Label (367,6 96x32), "Уставки"
    Label (227,6 123x32), "Актуальные"
END_VISUALIZATION

// Device/Application/Visu/DlgPids
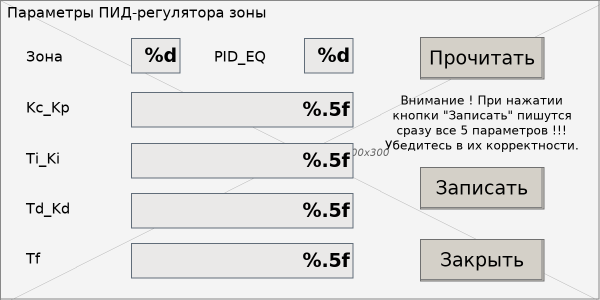
VISUALIZATION DlgPids  // 600x300
VAR_IN_OUT
	bDialogVar	: BOOL;
END_VAR
    Image (0,0 608x305), image: ImagePool.Dialog_win_7_600x300
    Button (420,37 124x42), "Прочитать"
        OnMouseClick: execute { Dvp.pid_read:=TRUE; }
    Button (420,239 124x42), "Закрыть"
        OnMouseClick:  Dialog=DlgPids, Result=OK, NumpadKeypadSet=True
    Label (4,3 296x19), "Параметры ПИД-регулятора зоны"
    Label (23,98 62x19), "Kc_Kp"
    RoundedRectangle (131,92 222x35), "%.5f", text variable: Dvp.Pids[Dvp.pid_index].Kc_Kp
        OnMouseClick: write the text variable via VisuDialogs.Numpad, min 0, max 1000, title "Пропорциональная часть"
    Label (23,149 62x19), "Ti_Ki"
    RoundedRectangle (131,143 222x35), "%.5f", text variable: Dvp.Pids[Dvp.pid_index].Ti_Ki
        OnMouseClick: write the text variable via VisuDialogs.Numpad, min 0, max 1000000, title "Интегральная часть"
    Label (23,199 62x19), "Td_Kd"
    RoundedRectangle (131,193 222x35), "%.5f", text variable: Dvp.Pids[Dvp.pid_index].Td_Kd
        OnMouseClick: write the text variable via VisuDialogs.Numpad, min 0, max 1000, title "Дифференциальная часть"
    RoundedRectangle (131,38 49x35), "%d", text variable: Dvp.zone_index
    Label (23,47 62x19), "Зона"
    Button (420,167 124x42), "Записать"
        OnMouseClick:  Dialog=DlgConfirm, Parameters={bDialogVar: Dvp.pid_write}, Selected={1: }, OpenModal=True, OpenCentered=True
    RoundedRectangle (304,38 49x35), "%d", text variable: Dvp.Pids[Dvp.pid_index].formula
        OnMouseClick: write the text variable via VisuDialogs.Numpad, min 0, max 1, format "Формула ПИД"
    Label (211,47 83x19), "PID_EQ"
    Label (23,249 62x19), "Tf"
    RoundedRectangle (131,243 222x35), "%.5f", text variable: Dvp.Pids[Dvp.pid_index].Tf
        OnMouseClick: write the text variable via VisuDialogs.Numpad, title "Пост.времени дифференцирования"
    Label (389,92 186x79), "Внимание ! При нажатии кнопки "Записать" пишутся сразу все 5 параметров !!! Убедитесь в их корректности."
END_VISUALIZATION

// Device/Application/Visu/VIS_SETTS_1
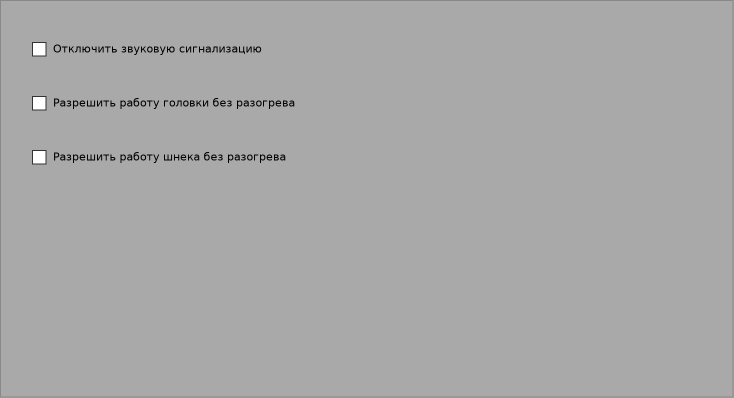
VISUALIZATION VIS_SETTS_1  // 734x398
    Checkbox (30,28 412x42), "Отключить звуковую сигнализацию", variable: Setts.otkl_alarm_zvuk
    Checkbox (30,82 412x42), "Разрешить работу головки без разогрева", variable: Setts.use_servo_without_temp
    Checkbox (30,136 412x42), "Разрешить работу шнека без разогрева", variable: Setts.use_shnek_without_temp
END_VISUALIZATION

// Device/Application/Visu/VIS_SETTS_2
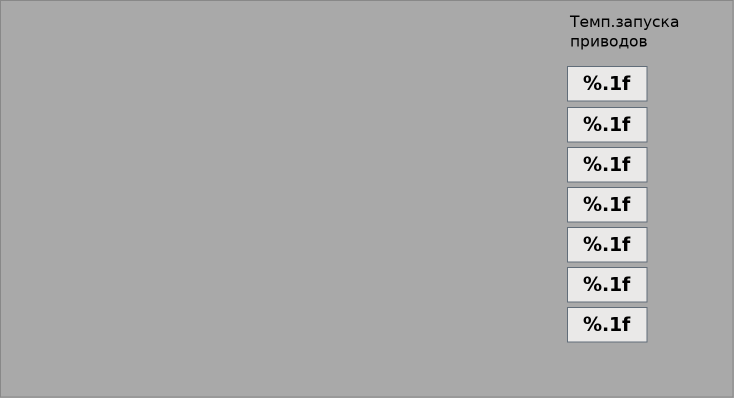
VISUALIZATION VIS_SETTS_2  // 734x398
    Label (567,11 119x45), "Темп.запуска приводов"
    RoundedRectangle (567,66 80x35), "%.1f", text variable: Setts.T_ZAP[0]
        OnMouseClick: write the text variable via VisuDialogs.Numpad, min 160, max 180
    RoundedRectangle (567,187 80x35), "%.1f", text variable: Setts.T_ZAP[3]
        OnMouseClick: write the text variable via VisuDialogs.Numpad, min 300, max 350
    RoundedRectangle (567,227 80x35), "%.1f", text variable: Setts.T_ZAP[4]
        OnMouseClick: write the text variable via VisuDialogs.Numpad, min 220, max 260
    RoundedRectangle (567,267 80x35), "%.1f", text variable: Setts.T_ZAP[5]
        OnMouseClick: write the text variable via VisuDialogs.Numpad, min 230, max 280
    RoundedRectangle (567,307 80x35), "%.1f", text variable: Setts.T_ZAP[6]
        OnMouseClick: write the text variable via VisuDialogs.Numpad, min 230, max 280
    RoundedRectangle (567,147 80x35), "%.1f", text variable: Setts.T_ZAP[2]
        OnMouseClick: write the text variable via VisuDialogs.Numpad, min 300, max 340
    RoundedRectangle (567,107 80x35), "%.1f", text variable: Setts.T_ZAP[1]
        OnMouseClick: write the text variable via VisuDialogs.Numpad, min 310, max 330
END_VISUALIZATION

// Device/Application/Visu/VIS_SETTS_3
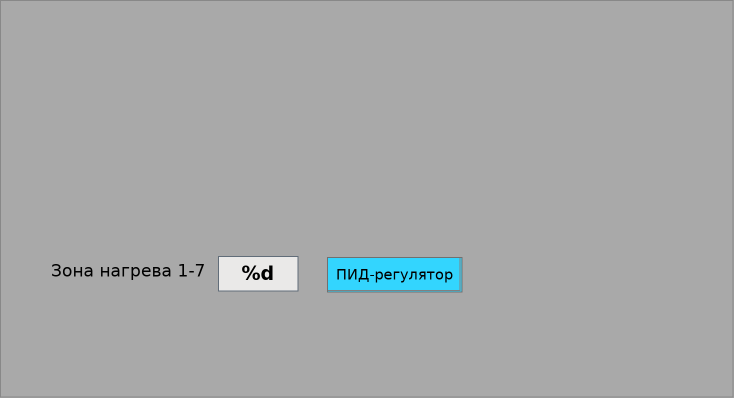
VISUALIZATION VIS_SETTS_3  // 734x398
    Label (48,259 166x28), "Зона нагрева 1-7"
    Button (327,257 135x35), "ПИД-регулятор"
        OnMouseClick:  Dialog=DlgPids, Parameters={bDialogVar: b_dialog}, Selected={1: }, OpenModal=True, OpenCentered=True
    RoundedRectangle (218,256 80x35), "%d", text variable: Dvp.zone_index
        OnMouseClick: write the text variable via VisuDialogs.Numpad, min 1, max 7, title "Введите зону нагрева 1-7"
END_VISUALIZATION

(* text list AsdaTextList (id | default)
  0 | Ожидание команды
  1 | Инициализация сервопривода
  2 | Поиск реперной точки (Homing)
  3 | Формирование каркаса
  4 | Операция отладочного перемещения
  5 | Операция задержки
  6 | Включение сервопривода
  7 | Экстренный останов
  8 | Отключение сервопривода
  9 | Установка параметров сервопривода
  10 | Обработка ошибки
  11 | Перемещение в реперную точку
  12 | Ожидание соединения
   |  *)

(* text list AG_DVP (id | default)
  8 | Каретка в крайнем положении
  7 | Превышено время возврата каретки на исходный концевик
  6 | Превышено время схода каретки с исходного концевика
  5 | Превышено время движения ножа
  4 | Превышено время схода ножа с исходного концевика
  3 | Превышено время движения зажима
  2 | Нож не на исходном концевике
  1 | Зажим не на исходном концевике
  0 | Каретка не на исходном концевике
   |  *)

(* text list DvpTextList (id | default)
  0 | Система в исходном состоянии
  1 | Система в режиме РАЗОГРЕВ
  2 | Система в рабочем состоянии
  3 | Система в режиме выгона массы
   |  *)

(* text list AG_CONNECT (id | default)
  4 | Нет соединения с Чиллером
  3 | Нет соединения с ПЧВ тянущего устройства
  2 | Нет соединения с ПЧВ шнека
  1 | Нет соединения с контроллером DVP
  0 | Нет соединение с сервоприводом ASDA-A2
   |  *)

(* text list MSGS (id | default)
  5 | 
  4 | Низкое давление воздуха !!!
  3 | Низкий уровень сырья в бункере !!!
  2 | Выведите бункер !!!
  1 | Бункер выведен !!!
  0 | Система вышла на режим !
   |  *)

(* text list AG_AVAR (id | default)
  4 | 
  3 | Низкая температура одной из зон
  2 | Превышена температура одной из зон
  1 | Температура одной из зон ниже температуры запуска привода
  0 | Превышена критическая температура одной из зон
   |  *)

(* text list AG_DEV (id | default)
  15 | Авария Чиллера - ALARM_3
  14 | Авария Чиллера - ALARM_2
  13 | Авария Чиллера
  12 | Перегрев ПЧВ тянущего устройства
  11 | Предел по току ПЧВ тянущего устройства
  10 | Аварийный сигнал ПЧВ тянущего устройства
  9 | Перегреве ПЧВ шнека
  8 | Предел по току ПЧВ шнека
  7 | Аварийный сигнал ПЧВ шнека
  6 | Тестовая ошибка
  5 | Превышено время операции отладки
  4 | РЕЗЕРВ АВАРИИ
  3 | Превышено время операции HOMING
  2 | Ошибка инициализации Р2-30 или Р3-06
  1 | Сигнал предупреждения от сервопривода
  0 | Сигнал аварии от сервопривода
   |  *)
